FUNCTION_BLOCK SET_AT_INDEX (* Set value of array at given index. Data types of value to be set must correspond to the array data type. Data type of resulting output array must correspond to input array data type. *)
  PACKAGE eclipse4diac::convert;
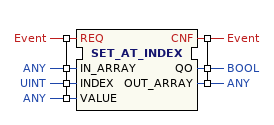
  EVENT_INPUT
    REQ WITH IN_ARRAY, INDEX, VALUE; (* Service Request *)
  END_EVENT
  EVENT_OUTPUT
    CNF WITH QO, OUT_ARRAY; (* Confirmation of Requested Service *)
  END_EVENT
  VAR_INPUT
    IN_ARRAY : ANY; (* input array *)
    INDEX : UINT; (* index to fetch value from *)
    VALUE : ANY; (* value to be copied to given index *)
  END_VAR
  VAR_OUTPUT
    QO : BOOL; (* Event Output Qualifier *)
    OUT_ARRAY : ANY; (* resulting array after set *)
  END_VAR
END_FUNCTION_BLOCK
